TYPE ST_ClampingMotionConfig :
STRUCT
    fVelocity : LREAL;
    fAcceleration : LREAL;
    fDeceleration : LREAL;
    fPositionTolerance : LREAL;
    tMoveTimeout : TIME;
END_STRUCT
END_TYPE

(* stored: Version 1.1.0.1, ProductVersion 3.1.4026.20
   DUT ST_ClampingMotionConfig: Id {0040004b-953c-4761-8d6b-16a053943107} *)
